Fanuc TP program (LS listing): S101_DR_T18N50.LS

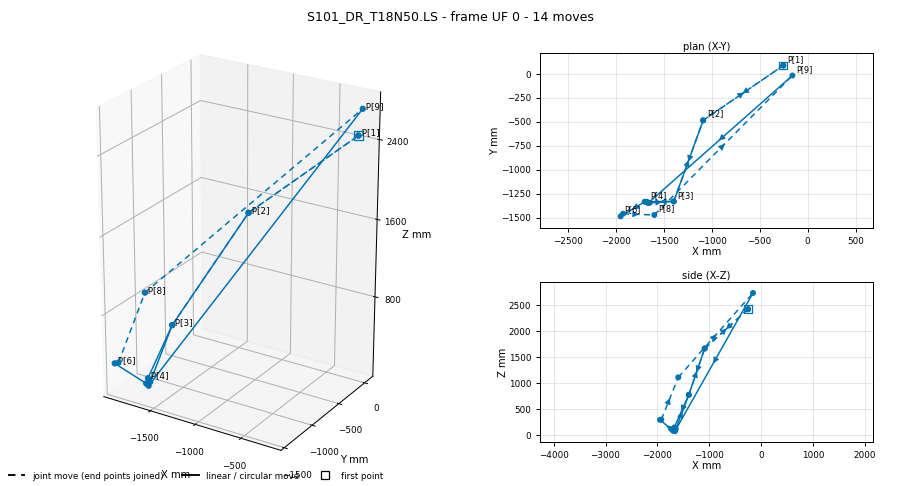
[picture p0: tool path of S101_DR_T18N50.LS in frame UF 0, 14 of 14 moves have a stored position in this frame; points joined in program order, loops and branches not executed]
/PROG  S101_DR_T18N50
/ATTR
OWNER		= MNEDITOR;
COMMENT		= "TL DRP TYP1 N50";
PROG_SIZE	= 3619;
CREATE		= DATE 19-07-31  TIME 09:46:40;
MODIFIED	= DATE 19-09-09  TIME 11:04:08;
FILE_NAME	= S101_DR_;
VERSION		= 0;
LINE_COUNT	= 124;
MEMORY_SIZE	= 4011;
PROTECT		= READ_WRITE;
STORAGE		= SHADOW;
TCD:  STACK_SIZE	= 0,
      TASK_PRIORITY	= 50,
      TIME_SLICE	= 0,
      BUSY_LAMP_OFF	= 0,
      ABORT_REQUEST	= 0,
      PAUSE_REQUEST	= 0;
DEFAULT_GROUP	= 1,*,*,*,*;
CONTROL_CODE	= 00000000 00000000;
/APPL
/MN
   1:  !******************************** ;
   2:  ! PATH - drop tool into N1=STA 70 ;
   3:  !******************************** ;
   4:  !* Robot ID: XXXXXR02B1 ;
   5:  !*    F-19XXXX ;
   6:  !* Line: XXXXXXXX ;
   7:  !* Platform: XX ;
   8:  !* Tool ID: TOOL xx ;
   9:  !* Program: S001_DR_TxxN3_R02 ;
  10:  !* Application: TOOL DROP ;
  11:  !******************************** ;
  12:  ! Author- Esys Automation ;
  13:  !******************************** ;
  14:   ;
  15:  !++++++++++++++++++++++++++++++++ ;
  16:  !ASSIGN PROGRAM PATH VALUES ;
  17:  !-------------------------------- ;
  18:  !Set Robot Tool and World UFrame ;
  19:  UTOOL_NUM=2 ;
  20:  UFRAME_NUM=0 ;
  21:  !++++++++++++++++++++++++++++++++ ;
  22:   ;
  23:  !******************************** ;
  24:  !BEGINNING OF PROGRAM PATH ;
  25:  !MOVE TO NEST 1 TOOL DROP ;
  26:  !******************************** ;
  27:   ;
  28:  !-------------------------------- ;
  29:  LBL[10:MOVE TO TL DRP] ;
  30:   ;
  31:  SET SEGMENT(50) ;
  32:  !SEG(50), Approach Tool Drop ;
  33:   ;
  34:J P[1] 100% CNT100    ;
  35:   ;
  36:J P[2] 100% CNT100    ;
  37:   ;
  38:L P[3:Tool-Pick-Pounce] 3000mm/sec CNT100    ;
  39:   ;
  40:L P[4] 300mm/sec CNT25    ;
  41:   ;
  42:L P[11] 50mm/sec FINE    ;
  43:   ;
  44:   ;
  45:  !-------------------------------- ;
  46:  LBL[20:UNLATCH TOOL] ;
  47:  UNLATCH TOOL    ;
  48:   ;
  49:  !ADD DISCONNECT COMMANDS ;
  50:  !ADD ALL EOAT DEVICES ;
  51:  !CALL EN_ARON(x) ;
  52:  !x = EOAT ENET Node # ;
  53:   ;
  54:  !If TL UNL Pass, Return Home ;
  55:  !If TL UNL Fail, Latch Tool, ;
  56:  !  MHFault, and Return Home ;
  57:  IF R[170]=1,JMP LBL[30] ;
  58:   ;
  59:  SELECT R[168]=7,JMP LBL[80] ;
  60:         ELSE,JMP LBL[99] ;
  61:   ;
  62:  !-------------------------------- ;
  63:  LBL[30:COMPLETE PATH] ;
  64:  !TL DRP COMPLETE. MOVE AWAY ;
  65:  !AND RETURN HOME ;
  66:   ;
  67:  !Set ATI Tool and World Frame ;
  68:  PAYLOAD[1] ;
  69:  UTOOL_NUM=14 ;
  70:  UFRAME_NUM=0 ;
  71:   ;
  72:  SET SEGMENT(51) ;
  73:  !SEG(51), Tool Drop Depart ;
  74:   ;
  75:L P[6:Tool-Pick-Apr] 50mm/sec FINE    ;
  76:   ;
  77:L P[7] 2000mm/sec CNT100    ;
  78:   ;
  79:J P[8] 100% CNT100    ;
  80:J P[9] 100% CNT100    ;
  81:   ;
  82:  ! Move To Home ;
  83:  JMP LBL[100] ;
  84:   ;
  85:  !-------------------------------- ;
  86:  LBL[80:UNLATCH FAULT] ;
  87:  !MOVE BACK TO HOME WITH TOOL ;
  88:  !on Reverse Path before Tool Drop ;
  89:   ;
  90:  !Set Payload= ATI ;
  91:  R[221]=1    ;
  92:  PAYLOAD[R[221]] ;
  93:  UFRAME_NUM=0 ;
  94:  UTOOL_NUM=2 ;
  95:   ;
  96:  LATCH TOOL    ;
  97:   ;
  98:L P[5:DROP_T07_N050] 50mm/sec FINE    ;
  99:   ;
 100:L P[10:Tool-Pick-Dep] 250mm/sec CNT25    ;
 101:   ;
 102:L P[3:Tool-Pick-Pounce] 2000mm/sec CNT100    ;
 103:   ;
 104:J P[2] 100% CNT100    ;
 105:J P[1] 100% CNT100    ;
 106:   ;
 107:  SET SEGMENT(63) ;
 108:  !SEG(63), Robot Move to Home ;
 109:   ;
 110:  R[132]=0    ;
 111:  GO[71]=0 ;
 112:   ;
 113:  ! Move To Home ;
 114:  JMP LBL[100] ;
 115:   ;
 116:  !-------------------------------- ;
 117:  LBL[99:ABORT PROGRAM] ;
 118:  MESSAGE[...] ;
 119:  MESSAGE[ABORT PROGRAM] ;
 120:  ABORT ;
 121:   ;
 122:  !-------------------------------- ;
 123:  LBL[100:END OF PROGRAM] ;
 124:  END ;
/POS
P[1]{
   GP1:
	UF : 0, UT : 2,		CONFIG : 'N U B, 0, 0, 0',
	X =  -253.309  mm,	Y =    88.384  mm,	Z =  2426.870  mm,
	W =   -93.331 deg,	P =     1.054 deg,	R =   122.429 deg
};
P[2]{
   GP1:
	UF : 0, UT : 2,		CONFIG : 'N U T, 0, 0, 0',
	X = -1089.020  mm,	Y =  -483.560  mm,	Z =  1671.145  mm,
	W =  -119.401 deg,	P =    -2.194 deg,	R =   112.860 deg
};
P[3:"Tool-Pick-Pounce"]{
   GP1:
	UF : 0, UT : 2,		CONFIG : 'N U T, 0, 0, 0',
	X = -1395.673  mm,	Y = -1328.706  mm,	Z =   776.338  mm,
	W =  -160.646 deg,	P =      .808 deg,	R =    90.629 deg
};
P[4]{
   GP1:
	UF : 0, UT : 2,		CONFIG : 'N U T, 0, 0, 0',
	X = -1677.509  mm,	Y = -1331.848  mm,	Z =   147.950  mm,
	W =  -161.318 deg,	P =     -.096 deg,	R =    91.596 deg
};
P[5:"DROP_T07_N050"]{
   GP1:
	UF : 0, UT : 2,		CONFIG : 'N U T, 0, 0, 0',
	X = -1662.466  mm,	Y = -1345.853  mm,	Z =    77.286  mm,
	W =  -161.155 deg,	P =     1.553 deg,	R =    88.655 deg
};
P[6:"Tool-Pick-Apr"]{
   GP1:
	UF : 0, UT : 14,		CONFIG : 'N U T, 0, 0, 0',
	X = -1949.940  mm,	Y = -1484.415  mm,	Z =   296.524  mm,
	W =  -159.789 deg,	P =     -.468 deg,	R =    92.970 deg
};
P[7]{
   GP1:
	UF : 0, UT : 14,		CONFIG : 'N U T, 0, 0, 0',
	X = -1924.475  mm,	Y = -1457.268  mm,	Z =   300.440  mm,
	W =  -159.530 deg,	P =      .503 deg,	R =    90.944 deg
};
P[8]{
   GP1:
	UF : 0, UT : 14,		CONFIG : 'N U T, 0, 0, 0',
	X = -1598.294  mm,	Y = -1470.396  mm,	Z =  1114.792  mm,
	W =  -159.094 deg,	P =      .421 deg,	R =    91.998 deg
};
P[9]{
   GP1:
	UF : 0, UT : 14,		CONFIG : 'N U B, 0, 0, 0',
	X =  -158.400  mm,	Y =   -15.894  mm,	Z =  2741.103  mm,
	W =   -91.792 deg,	P =     -.357 deg,	R =   122.600 deg
};
P[10:"Tool-Pick-Dep"]{
   GP1:
	UF : 0, UT : 2,		CONFIG : 'N U T, 0, 0, 0',
	X = -1646.146  mm,	Y = -1343.035  mm,	Z =   119.837  mm,
	W =  -161.370 deg,	P =      .449 deg,	R =    89.746 deg
};
P[11]{
   GP1:
	UF : 0, UT : 2,		CONFIG : 'N U T, 0, 0, 0',
	X = -1698.588  mm,	Y = -1332.323  mm,	Z =    85.534  mm,
	W =  -161.320 deg,	P =     -.097 deg,	R =    91.597 deg
};
/END
